SUBAPPLICATION Abscheider (* Subapplication Type *)
  (* Standard: 61499-2 *)
  (* Version 1.0, 2023-01-29, Franz *)
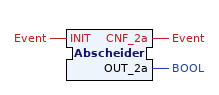
  EVENT_INPUT
    INIT;
  END_EVENT
  EVENT_OUTPUT
    CNF_2a;
  END_EVENT
  VAR_OUTPUT
    OUT_2a : BOOL;
  END_VAR
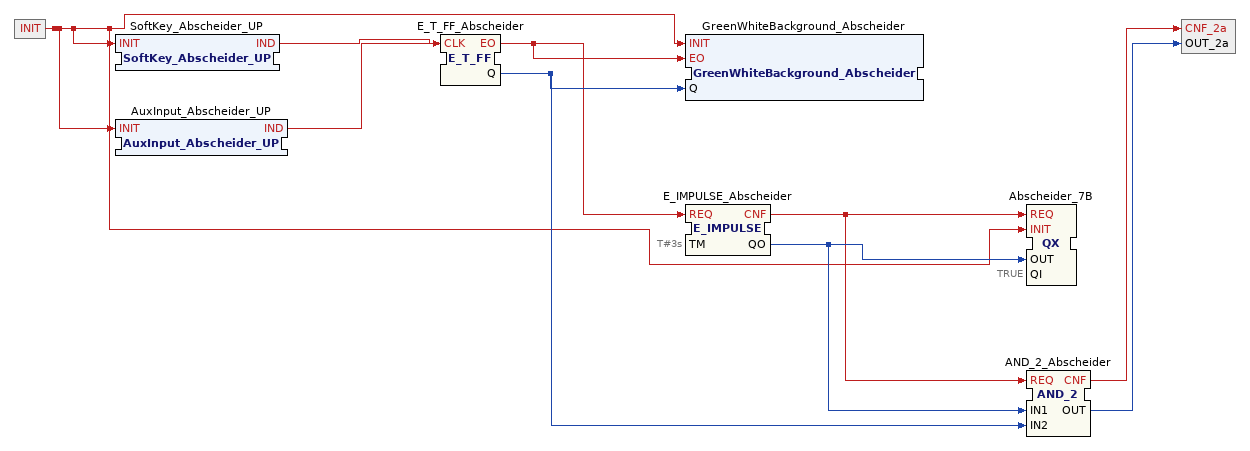
  FBS
    AND_2_Abscheider : AND_2;
    E_T_FF_Abscheider : E_T_FF;
    Abscheider_7B : QX(QI := TRUE);
    E_IMPULSE_Abscheider : E_IMPULSE(TM := T#3s);
  END_FBS
  SUBAPPS
    GreenWhiteBackground_Abscheider : GreenWhiteBackground_Abscheider;
    AuxInput_Abscheider_UP : AuxInput_Abscheider_UP;
    SoftKey_Abscheider_UP : SoftKey_Abscheider_UP;
  END_SUBAPPS
  EVENT_CONNECTIONS
    E_IMPULSE_Abscheider.CNF TO AND_2_Abscheider.REQ;
    E_T_FF_Abscheider.EO TO E_IMPULSE_Abscheider.REQ;
    E_IMPULSE_Abscheider.CNF TO Abscheider_7B.REQ;
    AND_2_Abscheider.CNF TO CNF_2a;
    INIT TO Abscheider_7B.INIT;
    INIT TO GreenWhiteBackground_Abscheider.INIT;
    E_T_FF_Abscheider.EO TO GreenWhiteBackground_Abscheider.EO;
    INIT TO AuxInput_Abscheider_UP.INIT;
    AuxInput_Abscheider_UP.IND TO E_T_FF_Abscheider.CLK;
    INIT TO SoftKey_Abscheider_UP.INIT;
    SoftKey_Abscheider_UP.IND TO E_T_FF_Abscheider.CLK;
  END_CONNECTIONS
  DATA_CONNECTIONS
    E_IMPULSE_Abscheider.QO TO AND_2_Abscheider.IN1;
    E_T_FF_Abscheider.Q TO AND_2_Abscheider.IN2;
    E_IMPULSE_Abscheider.QO TO Abscheider_7B.OUT;
    AND_2_Abscheider.OUT TO OUT_2a;
    E_T_FF_Abscheider.Q TO GreenWhiteBackground_Abscheider.Q;
  END_CONNECTIONS
END_SUBAPPLICATION
